// Mitsubishi GX Works2 project: 카운터플리커   PLC: Q03UDV

PROGRAM MAIN
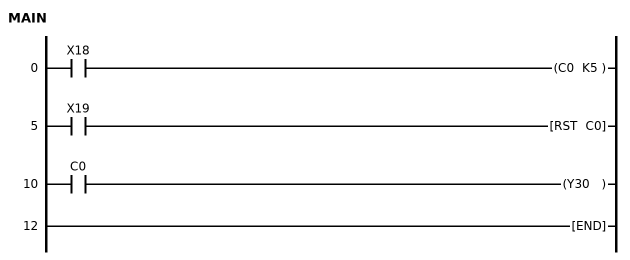
0     LD      X18
      OUT     C0 K5
5     LD      X19
      RST     C0
10    LD      C0
      OUT     Y30
12    END
END_PROGRAM
